// Library/POUs/Read/MC_ReadToolData/Structures/ReadToolDataParCmd
{attribute 'pack_mode' := '1'} 
// ------------------------------------------------------------------------- 
//  SRCI Robot Library                                                
// ------------------------------------------------------------------------- 
//                                                                           
//  Object:      ReadToolDataParCmd                                       
//  Author:      Thorsten Brach                                                
//  Date:        2024-08-09
//
//  Description:                                              
//   
//                                                                           
//  Copyright: 
//    (C) 2024 Thorsten Brach. All rights reserved                                                                                                                                            
//             Licensed under the LGPL-3.0 license.
//                                                                           
//  Disclaimer:                                                                           
//    This project is provided without any guarantee and can be used for   
//    private and commercial purposes. Any use is at the user’s 
//    own risk and responsibility.
//
// -------------------------------------------------------------------------
TYPE ReadToolDataParCmd :
STRUCT
  /// Tool index
  /// • -1: Currently used tool on RC
  /// •  0: Flange -  Not possible to change
  /// • 1 (default)..254: Tool Frame
  ToolNo             : INT;
END_STRUCT
END_TYPE

// Library/POUs/Read/MC_ReadToolData/Structures/ReadToolDataRecvData
{attribute 'pack_mode' := '1'} 
// ------------------------------------------------------------------------- 
//  SRCI Robot Library                                                
// ------------------------------------------------------------------------- 
//                                                                           
//  Object:      ReadToolDataRecvData                                       
//  Author:      Thorsten Brach                                                
//  Date:        2024-08-09
//
//  Description:                                              
//   
//                                                                           
//  Copyright: 
//    (C) 2024 Thorsten Brach. All rights reserved                                                                                                                                            
//             Licensed under the LGPL-3.0 license.
//                                                                           
//  Disclaimer:                                                                           
//    This project is provided without any guarantee and can be used for   
//    private and commercial purposes. Any use is at the user’s 
//    own risk and responsibility.
//
// -------------------------------------------------------------------------
TYPE ReadToolDataRecvData EXTENDS RspHeader :
STRUCT
  /// Reserve
  Reserve       : BYTE;
  /// Tool index
  ToolNoReturn  : USINT;
  /// Tool data (see chapter 5.5.6.3)
  ToolData      : ToolData;
  /// ToDo
  DataChanged   : BOOL;
END_STRUCT
END_TYPE

// Library/POUs/Read/MC_ReadToolData/Structures/ReadToolDataSendData
{attribute 'pack_mode' := '1'}
// ------------------------------------------------------------------------- 
//  SRCI Robot Library                                                
// ------------------------------------------------------------------------- 
//                                                                           
//  Object:      ReadToolDataSendData                                       
//  Author:      Thorsten Brach                                                
//  Date:        2024-08-09
//
//  Description:                                              
//   
//                                                                           
//  Copyright: 
//    (C) 2024 Thorsten Brach. All rights reserved                                                                                                                                            
//             Licensed under the LGPL-3.0 license.
//                                                                           
//  Disclaimer:                                                                           
//    This project is provided without any guarantee and can be used for   
//    private and commercial purposes. Any use is at the user’s 
//    own risk and responsibility.
//
// -------------------------------------------------------------------------
TYPE ReadToolDataSendData EXTENDS CmdHeader: 
STRUCT
  /// Tool index
  /// • -1: Currently used tool on RC
  /// •  0: Flange -  Not possible to change
  /// • 1 (default)..254: Tool Frame
  ToolNo             : INT;
END_STRUCT
END_TYPE

// Library/POUs/SearchHardstop/MC_SearchHardStop/Structures/SearchHardStopOutCmd
{attribute 'pack_mode' := '1'} 
// ------------------------------------------------------------------------- 
//  SRCI Robot Library                                                
// ------------------------------------------------------------------------- 
//                                                                           
//  Object:      SearchHardStopOutCmd                                       
//  Author:      Thorsten Brach                                                
//  Date:        2024-08-01
//
//  Description:                                              
//   
//                                                                           
//  Copyright: 
//    (C) 2024 Thorsten Brach. All rights reserved                                                                                                                                            
//             Licensed under the LGPL-3.0 license.
//                                                                           
//  Disclaimer:                                                                           
//    This project is provided without any guarantee and can be used for   
//    private and commercial purposes. Any use is at the user’s 
//    own risk and responsibility.
//
// -------------------------------------------------------------------------
TYPE SearchHardStopOutCmd :
STRUCT
  /// Distance-to-go of the current job.
  /// • -1: No valid value because move command is not yet active (valid values are pending) or not supported by RC
  /// • >0: Actual distance between current and target position
  /// •  0: Target position reached
  RemainingDistance  : REAL;
  /// Percentage of already traversed distance of current job.
  /// If not supported : • -1
  Progress           : REAL;
  /// The robot arm has detected an obstruction and stopped the movement
  InClamping         : BOOL;  
END_STRUCT
END_TYPE

// Library/POUs/SearchHardstop/MC_SearchHardStop/Structures/SearchHardStopParCmd
{attribute 'pack_mode' := '1'} 
// ------------------------------------------------------------------------- 
//  SRCI Robot Library                                                
// ------------------------------------------------------------------------- 
//                                                                           
//  Object:      SearchHardStopParCmd                                       
//  Author:      Thorsten Brach                                                
//  Date:        2024-08-01
//
//  Description:                                              
//   
//                                                                           
//  Copyright: 
//    (C) 2024 Thorsten Brach. All rights reserved                                                                                                                                            
//             Licensed under the LGPL-3.0 license.
//                                                                           
//  Disclaimer:                                                                           
//    This project is provided without any guarantee and can be used for   
//    private and commercial purposes. Any use is at the user’s 
//    own risk and responsibility.
//
// -------------------------------------------------------------------------
TYPE SearchHardStopParCmd :
STRUCT
  /// Absolute target coordinates in the selected coordinate system (see input parameters ToolNo and FrameNo)
  Position           : RobotCartesianPosition;
  /// Defines the type of collision detection, which parameter should be observed
  DetectionMode      : DetectionMode;
  /// Additional parameter for the detection of an end position. Defines the limits for seven joints, 
  /// where the robot stops when one of the limits is reached. Unit is depending on the "DetectionMode":
  /// • Torque (default) [Nm]  - Only positive values accepted
  /// • Force [N]              - Only positive values accepted
  /// • Electrical current [A] - Only positive values accepted
  /// • Following Error [mm]   - >0: Robot stops when the following error reached positive limit
  ///                          - <0: Robot stops when the following error reaches the negative limit
  DetectionVector    : ARRAY [0..5] OF REAL;
  /// TCP velocity in % of nominal velocity
  /// •  <0%: (default) - Use default velocity
  /// •   0%:           - Use internal minimal velocity
  /// • 100%:           - Use maximal reference velocity
  /// See chapter 5.5.7 Robot dynamics
  VelocityRate       : REAL;
  /// Acceleration for movement in % of nominal acceleration
  /// •  <0%: (default) - Use default acceleration
  /// •   0%:           - Use internal minimal acceleration
  /// • 100%:           - Use maximal reference acceleration
  /// See chapter 5.5.7 Robot dynamics
  AccelerationRate   : REAL;
  /// Deceleration for movement in % of nominal deceleration
  /// •  <0%: (default) - Use default deceleration 
  /// •   0%:           - Use internal minimal deceleration
  /// • 100%:           - Use maximal reference deceleration
  /// See chapter 5.5.7 Robot dynamics
  DecelerationRate   : REAL;
  /// Jerk of the movement in % of nominal jerk
  /// •  <0%: (default) - Use default jerk
  /// •   0%:           - Use internal minimal jerk
  /// • 100%:           - Use maximal reference jerk
  /// See chapter 5.5.7 Robot dynamics
  JerkRate           : REAL;
  /// Index of tool
  /// •      0: Flange (default)
  /// • 1..254: Tool frames
  ToolNo             : USINT;
  /// Index of frame
  /// •      0: WCS (default)
  /// • 1..254: User frames
  FrameNo            : USINT;
  /// Parameter to describe how the orientation axes (RX, RY, RZ) will be interpolated during the movement
  OriMode            : OriMode;
  /// Defines the usage of the config byte inside the position according to Table 6-238
  ConfigMode         : ArmConfigParameter;
  /// Defines the usage of the TurnNumber byte inside the position.
  TurnMode           : TurnMode;
  /// Set TRUE to allow manipulation of this move command through superimposing functions.
  /// For more information see chapter 5.5.9.5
  Manipulation       : BOOL;
END_STRUCT
END_TYPE

// Library/POUs/SearchHardstop/MC_SearchHardStop/Structures/SearchHardStopRecvData
{attribute 'pack_mode' := '1'} 
// ------------------------------------------------------------------------- 
//  SRCI Robot Library                                                
// ------------------------------------------------------------------------- 
//                                                                           
//  Object:      SearchHardStopRecvData                                       
//  Author:      Thorsten Brach                                                
//  Date:        2024-08-01
//
//  Description:                                              
//   
//                                                                           
//  Copyright: 
//    (C) 2024 Thorsten Brach. All rights reserved                                                                                                                                            
//             Licensed under the LGPL-3.0 license.
//                                                                           
//  Disclaimer:                                                                           
//    This project is provided without any guarantee and can be used for   
//    private and commercial purposes. Any use is at the user’s 
//    own risk and responsibility.
//
// -------------------------------------------------------------------------
TYPE SearchHardStopRecvData EXTENDS RspHeader :
STRUCT
  /// Percentage of already traversed distance of current job.
  /// If not supported : • -1
  Progress           : UINT;
  /// Distance-to-go of the current job.
  /// • -1: No valid value because move command is not yet active (valid values are pending) or not supported by RC
  /// • >0: Actual distance between current and target position
  /// •  0: Target position reached
  RemainingDistance  : REAL;
  /// The robot arm has detected an obstruction and stopped the movement
  InClamping         : BOOL;  
END_STRUCT
END_TYPE

// Library/POUs/SearchHardstop/MC_SearchHardStop/Structures/SearchHardStopSendData
{attribute 'pack_mode' := '1'}
// ------------------------------------------------------------------------- 
//  SRCI Robot Library                                                
// ------------------------------------------------------------------------- 
//                                                                           
//  Object:      SearchHardStopSendData                                       
//  Author:      Thorsten Brach                                                
//  Date:        2024-08-01
//
//  Description:                                              
//   
//                                                                           
//  Copyright: 
//    (C) 2024 Thorsten Brach. All rights reserved                                                                                                                                            
//             Licensed under the LGPL-3.0 license.
//                                                                           
//  Disclaimer:                                                                           
//    This project is provided without any guarantee and can be used for   
//    private and commercial purposes. Any use is at the user’s 
//    own risk and responsibility.
//
// -------------------------------------------------------------------------
TYPE SearchHardStopSendData EXTENDS CmdHeader: 
STRUCT
  /// TCP velocity in % of nominal velocity
  /// •  <0%: (default) - Use default velocity
  /// •   0%:           - Use internal minimal velocity
  /// • 100%:           - Use maximal reference velocity
  /// See chapter 5.5.7 Robot dynamics
  VelocityRate       : UINT;
  /// Acceleration for movement in % of nominal acceleration
  /// •  <0%: (default) - Use default acceleration
  /// •   0%:           - Use internal minimal acceleration
  /// • 100%:           - Use maximal reference acceleration
  /// See chapter 5.5.7 Robot dynamics
  AccelerationRate   : UINT;
  /// Deceleration for movement in % of nominal deceleration
  /// •  <0%: (default) - Use default deceleration 
  /// •   0%:           - Use internal minimal deceleration
  /// • 100%:           - Use maximal reference deceleration
  /// See chapter 5.5.7 Robot dynamics
  DecelerationRate   : UINT;
  /// Jerk of the movement in % of nominal jerk
  /// •  <0%: (default) - Use default jerk
  /// •   0%:           - Use internal minimal jerk
  /// • 100%:           - Use maximal reference jerk
  /// See chapter 5.5.7 Robot dynamics
  JerkRate           : UINT;
  /// Index of tool
  /// •      0: Flange (default)
  /// • 1..254: Tool frames
  ToolNo             : USINT;
  /// Index of frame
  /// •      0: WCS (default)
  /// • 1..254: User frames
  FrameNo            : USINT;
  /// Absolute target coordinates in the selected coordinate system (see input parameters ToolNo and FrameNo)
  Position           : RobotCartesianPosition;
  /// Parameter to describe how the orientation axes (RX, RY, RZ) will be interpolated during the movement
  OriMode            : USINT;
  /// Defines the type of collision detection, which parameter should be observed
  DetectionMode      : USINT;
  /// Set TRUE to allow manipulation of this move command through superimposing functions.
  /// For more information see chapter 5.5.9.5
  Manipulation       : BOOL;
  /// Reserve
  Reserve            : BYTE;
  /// Additional parameter for the detection of an end position. Defines the limits for seven joints, 
  /// where the robot stops when one of the limits is reached. Unit is depending on the "DetectionMode":
  /// • Torque (default) [Nm]  - Only positive values accepted
  /// • Force [N]              - Only positive values accepted
  /// • Electrical current [A] - Only positive values accepted
  /// • Following Error [mm]   - >0: Robot stops when the following error reached positive limit
  ///                          - <0: Robot stops when the following error reaches the negative limit
  DetectionVector    : ARRAY [0..5] OF REAL;
  /// Defines the usage of the config byte inside the position according to Table 6-238
  ConfigMode         : ARRAY [0..1] OF BYTE;
  /// Defines the usage of the TurnNumber byte inside the position.
  TurnMode           : USINT;
END_STRUCT
END_TYPE

// Library/POUs/SearchHardstop/MC_SearchHardStopJ/Structures/SearchHardStopJOutCmd
{attribute 'pack_mode' := '1'} 
// ------------------------------------------------------------------------- 
//  SRCI Robot Library                                                
// ------------------------------------------------------------------------- 
//                                                                           
//  Object:      SearchHardStopOutCmd                                       
//  Author:      Thorsten Brach                                                
//  Date:        2024-08-01
//
//  Description:                                              
//   
//                                                                           
//  Copyright: 
//    (C) 2024 Thorsten Brach. All rights reserved                                                                                                                                            
//             Licensed under the LGPL-3.0 license.
//                                                                           
//  Disclaimer:                                                                           
//    This project is provided without any guarantee and can be used for   
//    private and commercial purposes. Any use is at the user’s 
//    own risk and responsibility.
//
// -------------------------------------------------------------------------
TYPE SearchHardStopJOutCmd :
STRUCT
  /// Distance-to-go of the current job.
  /// • -1: No valid value because move command is not yet active (valid values are pending) or not supported by RC
  /// • >0: Actual distance between current and target position
  /// •  0: Target position reached
  RemainingDistance  : REAL;
  /// Percentage of already traversed distance of current job.
  /// If not supported : • -1
  Progress           : REAL;
  /// The robot arm has detected an obstruction and stopped the movement
  InClamping         : BOOL;  
END_STRUCT
END_TYPE

// Library/POUs/SearchHardstop/MC_SearchHardStopJ/Structures/SearchHardStopJParCmd
{attribute 'pack_mode' := '1'} 
// ------------------------------------------------------------------------- 
//  SRCI Robot Library                                                
// ------------------------------------------------------------------------- 
//                                                                           
//  Object:      SearchHardStopParCmd                                       
//  Author:      Thorsten Brach                                                
//  Date:        2024-08-01
//
//  Description:                                              
//   
//                                                                           
//  Copyright: 
//    (C) 2024 Thorsten Brach. All rights reserved                                                                                                                                            
//             Licensed under the LGPL-3.0 license.
//                                                                           
//  Disclaimer:                                                                           
//    This project is provided without any guarantee and can be used for   
//    private and commercial purposes. Any use is at the user’s 
//    own risk and responsibility.
//
// -------------------------------------------------------------------------
TYPE SearchHardStopJParCmd :
STRUCT
  /// Absolute end position of the robot in Joint position.
  JointPosition      : RobotJointPosition;
  /// Defines the type of collision detection, which parameter should be observed
  DetectionMode      : DetectionMode;
  /// Additional parameter for the detection of an end position. Defines the limits for seven joints, 
  /// where the robot stops when one of the limits is reached. Unit is depending on the "DetectionMode":
  /// • Torque (default) [Nm]  - Only positive values accepted
  /// • Force [N]              - Only positive values accepted
  /// • Electrical current [A] - Only positive values accepted
  /// • Following Error [mm]   - >0: Robot stops when the following error reached positive limit
  ///                          - <0: Robot stops when the following error reaches the negative limit
  DetectionVector    : ARRAY [0..5] OF REAL;
  /// TCP velocity in % of nominal velocity
  /// •  <0%: (default) - Use default velocity
  /// •   0%:           - Use internal minimal velocity
  /// • 100%:           - Use maximal reference velocity
  /// See chapter 5.5.7 Robot dynamics
  VelocityRate       : REAL;
  /// Acceleration for movement in % of nominal acceleration
  /// •  <0%: (default) - Use default acceleration
  /// •   0%:           - Use internal minimal acceleration
  /// • 100%:           - Use maximal reference acceleration
  /// See chapter 5.5.7 Robot dynamics
  AccelerationRate   : REAL;
  /// Deceleration for movement in % of nominal deceleration
  /// •  <0%: (default) - Use default deceleration 
  /// •   0%:           - Use internal minimal deceleration
  /// • 100%:           - Use maximal reference deceleration
  /// See chapter 5.5.7 Robot dynamics
  DecelerationRate   : REAL;
  /// Jerk of the movement in % of nominal jerk
  /// •  <0%: (default) - Use default jerk
  /// •   0%:           - Use internal minimal jerk
  /// • 100%:           - Use maximal reference jerk
  /// See chapter 5.5.7 Robot dynamics
  JerkRate           : REAL;
  /// Index of tool
  /// •      0: Flange (default)
  /// • 1..254: Tool frames
  ToolNo             : USINT;
  /// Set TRUE to allow manipulation of this move command through superimposing functions.
  /// For more information see chapter 5.5.9.5
  Manipulation       : BOOL;
END_STRUCT
END_TYPE

// Library/POUs/SearchHardstop/MC_SearchHardStopJ/Structures/SearchHardStopJRecvData
{attribute 'pack_mode' := '1'} 
// ------------------------------------------------------------------------- 
//  SRCI Robot Library                                                
// ------------------------------------------------------------------------- 
//                                                                           
//  Object:      SearchHardStopRecvData                                       
//  Author:      Thorsten Brach                                                
//  Date:        2024-08-01
//
//  Description:                                              
//   
//                                                                           
//  Copyright: 
//    (C) 2024 Thorsten Brach. All rights reserved                                                                                                                                            
//             Licensed under the LGPL-3.0 license.
//                                                                           
//  Disclaimer:                                                                           
//    This project is provided without any guarantee and can be used for   
//    private and commercial purposes. Any use is at the user’s 
//    own risk and responsibility.
//
// -------------------------------------------------------------------------
TYPE SearchHardStopJRecvData EXTENDS RspHeader :
STRUCT
  /// Percentage of already traversed distance of current job.
  /// If not supported : • -1
  Progress           : UINT;
  /// Distance-to-go of the current job.
  /// • -1: No valid value because move command is not yet active (valid values are pending) or not supported by RC
  /// • >0: Actual distance between current and target position
  /// •  0: Target position reached
  RemainingDistance  : REAL;
  /// The robot arm has detected an obstruction and stopped the movement
  InClamping         : BOOL;  
END_STRUCT
END_TYPE

// Library/POUs/SearchHardstop/MC_SearchHardStopJ/Structures/SearchHardStopJSendData
{attribute 'pack_mode' := '1'}
// ------------------------------------------------------------------------- 
//  SRCI Robot Library                                                
// ------------------------------------------------------------------------- 
//                                                                           
//  Object:      SearchHardStopSendData                                       
//  Author:      Thorsten Brach                                                
//  Date:        2024-08-01
//
//  Description:                                              
//   
//                                                                           
//  Copyright: 
//    (C) 2024 Thorsten Brach. All rights reserved                                                                                                                                            
//             Licensed under the LGPL-3.0 license.
//                                                                           
//  Disclaimer:                                                                           
//    This project is provided without any guarantee and can be used for   
//    private and commercial purposes. Any use is at the user’s 
//    own risk and responsibility.
//
// -------------------------------------------------------------------------
TYPE SearchHardStopJSendData EXTENDS CmdHeader: 
STRUCT
  /// TCP velocity in % of nominal velocity
  /// •  <0%: (default) - Use default velocity
  /// •   0%:           - Use internal minimal velocity
  /// • 100%:           - Use maximal reference velocity
  /// See chapter 5.5.7 Robot dynamics
  VelocityRate       : UINT;
  /// Acceleration for movement in % of nominal acceleration
  /// •  <0%: (default) - Use default acceleration
  /// •   0%:           - Use internal minimal acceleration
  /// • 100%:           - Use maximal reference acceleration
  /// See chapter 5.5.7 Robot dynamics
  AccelerationRate   : UINT;
  /// Deceleration for movement in % of nominal deceleration
  /// •  <0%: (default) - Use default deceleration 
  /// •   0%:           - Use internal minimal deceleration
  /// • 100%:           - Use maximal reference deceleration
  /// See chapter 5.5.7 Robot dynamics
  DecelerationRate   : UINT;
  /// Jerk of the movement in % of nominal jerk
  /// •  <0%: (default) - Use default jerk
  /// •   0%:           - Use internal minimal jerk
  /// • 100%:           - Use maximal reference jerk
  /// See chapter 5.5.7 Robot dynamics
  JerkRate           : UINT;
  /// Absolute end position of the robot in Joint position.
  JointPosition      : RobotJointPosition;
  /// Parameter to describe how the orientation axes (RX, RY, RZ) will be interpolated during the movement
  OriMode            : USINT;
  /// Defines the type of collision detection, which parameter should be observed
  DetectionMode      : USINT;
  /// Set TRUE to allow manipulation of this move command through superimposing functions.
  /// For more information see chapter 5.5.9.5
  Manipulation       : BOOL;
  /// Reserve
  Reserve            : BYTE;
  /// Additional parameter for the detection of an end position. Defines the limits for seven joints, 
  /// where the robot stops when one of the limits is reached. Unit is depending on the "DetectionMode":
  /// • Torque (default) [Nm]  - Only positive values accepted
  /// • Force [N]              - Only positive values accepted
  /// • Electrical current [A] - Only positive values accepted
  /// • Following Error [mm]   - >0: Robot stops when the following error reached positive limit
  ///                          - <0: Robot stops when the following error reaches the negative limit
  DetectionVector    : ARRAY [0..5] OF REAL;
END_STRUCT
END_TYPE

// Library/POUs/Spline/MC_CreateSpline/Structures/CreateSplineOutCmd
{attribute 'pack_mode' := '1'} 
// ------------------------------------------------------------------------- 
//  SRCI Robot Library                                                
// ------------------------------------------------------------------------- 
//                                                                           
//  Object:      CreateSplineOutCmd                                       
//  Author:      Thorsten Brach                                                
//  Date:        2024-08-01
//
//  Description:                                              
//   
//                                                                           
//  Copyright: 
//    (C) 2024 Thorsten Brach. All rights reserved                                                                                                                                            
//             Licensed under the LGPL-3.0 license.
//                                                                           
//  Disclaimer:                                                                           
//    This project is provided without any guarantee and can be used for   
//    private and commercial purposes. Any use is at the user’s 
//    own risk and responsibility.
//
// -------------------------------------------------------------------------
TYPE CreateSplineOutCmd :
STRUCT
END_STRUCT
END_TYPE

// Library/POUs/Spline/MC_CreateSpline/Structures/CreateSplineParCmd
{attribute 'pack_mode' := '1'} 
// ------------------------------------------------------------------------- 
//  SRCI Robot Library                                                
// ------------------------------------------------------------------------- 
//                                                                           
//  Object:      CreateSplineParCmd                                       
//  Author:      Thorsten Brach                                                
//  Date:        2024-08-01
//
//  Description:                                              
//   
//                                                                           
//  Copyright: 
//    (C) 2024 Thorsten Brach. All rights reserved                                                                                                                                            
//             Licensed under the LGPL-3.0 license.
//                                                                           
//  Disclaimer:                                                                           
//    This project is provided without any guarantee and can be used for   
//    private and commercial purposes. Any use is at the user’s 
//    own risk and responsibility.
//
// -------------------------------------------------------------------------
TYPE CreateSplineParCmd :
STRUCT
  /// Define the method to calculate the path trajectory for the spline movement
  Mode            : SplineMode;
  /// Index of the spline trajectory to be created
  SplineID        : SINT;
  /// Contains all data relevant to the spline trajectory
  /// • Cartesian position
  /// • Coordinate systems
  /// • Dynamic parameters
  /// For more information refer to chapter 5.5.13.3
  SplineData      : ARRAY[1..RobotLibraryParameter.SPLINE_DATA_MAX] OF SplineData;
END_STRUCT
END_TYPE

// Library/POUs/Spline/MC_CreateSpline/Structures/CreateSplineRecvData
{attribute 'pack_mode' := '1'} 
// ------------------------------------------------------------------------- 
//  SRCI Robot Library                                                
// ------------------------------------------------------------------------- 
//                                                                           
//  Object:      CreateSplineRecvData                                       
//  Author:      Thorsten Brach                                                
//  Date:        2024-08-01
//
//  Description:                                              
//   
//                                                                           
//  Copyright: 
//    (C) 2024 Thorsten Brach. All rights reserved                                                                                                                                            
//             Licensed under the LGPL-3.0 license.
//                                                                           
//  Disclaimer:                                                                           
//    This project is provided without any guarantee and can be used for   
//    private and commercial purposes. Any use is at the user’s 
//    own risk and responsibility.
//
// -------------------------------------------------------------------------
TYPE CreateSplineRecvData EXTENDS RspHeader :
STRUCT
END_STRUCT
END_TYPE

// Library/POUs/Spline/MC_CreateSpline/Structures/CreateSplineSendData
{attribute 'pack_mode' := '1'}
// ------------------------------------------------------------------------- 
//  SRCI Robot Library                                                
// ------------------------------------------------------------------------- 
//                                                                           
//  Object:      CreateSplineSendData                                       
//  Author:      Thorsten Brach                                                
//  Date:        2024-08-01
//
//  Description:                                              
//   
//                                                                           
//  Copyright: 
//    (C) 2024 Thorsten Brach. All rights reserved                                                                                                                                            
//             Licensed under the LGPL-3.0 license.
//                                                                           
//  Disclaimer:                                                                           
//    This project is provided without any guarantee and can be used for   
//    private and commercial purposes. Any use is at the user’s 
//    own risk and responsibility.
//
// -------------------------------------------------------------------------
TYPE CreateSplineSendData EXTENDS CmdHeader: 
STRUCT
  /// Define the method to calculate the path trajectory for the spline movement
  Mode            : UINT;
  /// Index of the spline trajectory to be created
  SplineID        : SINT;
  /// Contains all data relevant to the spline trajectory
  /// • Cartesian position
  /// • Coordinate systems
  /// • Dynamic parameters
  /// For more information refer to chapter 5.5.13.3
  SplineData      : ARRAY[1..RobotLibraryParameter.SPLINE_DATA_MAX] OF SplineDataSend;
END_STRUCT
END_TYPE

// Library/POUs/Spline/MC_DeleteSpline/Structures/DeleteSplineOutCmd
{attribute 'pack_mode' := '1'} 
// ------------------------------------------------------------------------- 
//  SRCI Robot Library                                                
// ------------------------------------------------------------------------- 
//                                                                           
//  Object:      DeleteSplineOutCmd                                       
//  Author:      Thorsten Brach                                                
//  Date:        2024-08-01
//
//  Description:                                              
//   
//                                                                           
//  Copyright: 
//    (C) 2024 Thorsten Brach. All rights reserved                                                                                                                                            
//             Licensed under the LGPL-3.0 license.
//                                                                           
//  Disclaimer:                                                                           
//    This project is provided without any guarantee and can be used for   
//    private and commercial purposes. Any use is at the user’s 
//    own risk and responsibility.
//
// -------------------------------------------------------------------------
TYPE DeleteSplineOutCmd :
STRUCT
END_STRUCT
END_TYPE

// Library/POUs/Spline/MC_DeleteSpline/Structures/DeleteSplineParCmd
{attribute 'pack_mode' := '1'} 
// ------------------------------------------------------------------------- 
//  SRCI Robot Library                                                
// ------------------------------------------------------------------------- 
//                                                                           
//  Object:      DeleteSplineParCmd                                       
//  Author:      Thorsten Brach                                                
//  Date:        2024-08-01
//
//  Description:                                              
//   
//                                                                           
//  Copyright: 
//    (C) 2024 Thorsten Brach. All rights reserved                                                                                                                                            
//             Licensed under the LGPL-3.0 license.
//                                                                           
//  Disclaimer:                                                                           
//    This project is provided without any guarantee and can be used for   
//    private and commercial purposes. Any use is at the user’s 
//    own risk and responsibility.
//
// -------------------------------------------------------------------------
TYPE DeleteSplineParCmd :
STRUCT
  /// Index of the spline trajectory to be deleted
  SplineID        : SINT;
END_STRUCT
END_TYPE

// Library/POUs/Spline/MC_DeleteSpline/Structures/DeleteSplineRecvData
{attribute 'pack_mode' := '1'} 
// ------------------------------------------------------------------------- 
//  SRCI Robot Library                                                
// ------------------------------------------------------------------------- 
//                                                                           
//  Object:      DeleteSplineRecvData                                       
//  Author:      Thorsten Brach                                                
//  Date:        2024-08-01
//
//  Description:                                              
//   
//                                                                           
//  Copyright: 
//    (C) 2024 Thorsten Brach. All rights reserved                                                                                                                                            
//             Licensed under the LGPL-3.0 license.
//                                                                           
//  Disclaimer:                                                                           
//    This project is provided without any guarantee and can be used for   
//    private and commercial purposes. Any use is at the user’s 
//    own risk and responsibility.
//
// -------------------------------------------------------------------------
TYPE DeleteSplineRecvData EXTENDS RspHeader :
STRUCT
END_STRUCT
END_TYPE

// Library/POUs/Spline/MC_DeleteSpline/Structures/DeleteSplineSendData
{attribute 'pack_mode' := '1'}
// ------------------------------------------------------------------------- 
//  SRCI Robot Library                                                
// ------------------------------------------------------------------------- 
//                                                                           
//  Object:      DeleteSplineSendData                                       
//  Author:      Thorsten Brach                                                
//  Date:        2024-08-01
//
//  Description:                                              
//   
//                                                                           
//  Copyright: 
//    (C) 2024 Thorsten Brach. All rights reserved                                                                                                                                            
//             Licensed under the LGPL-3.0 license.
//                                                                           
//  Disclaimer:                                                                           
//    This project is provided without any guarantee and can be used for   
//    private and commercial purposes. Any use is at the user’s 
//    own risk and responsibility.
//
// -------------------------------------------------------------------------
TYPE DeleteSplineSendData EXTENDS CmdHeader: 
STRUCT
  /// Index of the spline trajectory to be deleted
  SplineID        : SINT;
END_STRUCT
END_TYPE

// Library/POUs/Spline/MC_DynamicSpline/Structures/DynamicSplineOutCmd
{attribute 'pack_mode' := '1'} 
// ------------------------------------------------------------------------- 
//  SRCI Robot Library                                                
// ------------------------------------------------------------------------- 
//                                                                           
//  Object:      DynamicSplineOutCmd                                       
//  Author:      Thorsten Brach                                                
//  Date:        2024-08-01
//
//  Description:                                              
//   
//                                                                           
//  Copyright: 
//    (C) 2024 Thorsten Brach. All rights reserved                                                                                                                                            
//             Licensed under the LGPL-3.0 license.
//                                                                           
//  Disclaimer:                                                                           
//    This project is provided without any guarantee and can be used for   
//    private and commercial purposes. Any use is at the user’s 
//    own risk and responsibility.
//
// -------------------------------------------------------------------------
TYPE DynamicSplineOutCmd :
STRUCT
  /// Distance-to-go of the current job.
  /// • -1: No valid value because move command is not yet active (valid values are pending) or not supported by RC
  /// • >0: Actual distance between current and target position
  /// •  0: Target position reached 
  RemainingDistance  : REAL;
  /// Percentage of already traversed distance of actual segment of spline trajectory.
  /// If not supported: -1
  SegmentProgress    : REAL;
  /// Number of buffered, consecutive segments of spline trajectory. 
  Buffered           : INT;
  /// Number of calculated, consecutive segments of spline trajectory. Already calculated segments can no longer be modified.
  Calculated         : INT;
  /// Index of the currently active segment of spline data set.
  ActiveIndex        : SINT;  
  /// Spline movement has been finished successfully. New SplineData will start a new spline movement.
  TrajectoryCompleted: BOOL;  
END_STRUCT
END_TYPE

// Library/POUs/Spline/MC_DynamicSpline/Structures/DynamicSplineParCmd
{attribute 'pack_mode' := '1'} 
// ------------------------------------------------------------------------- 
//  SRCI Robot Library                                                
// ------------------------------------------------------------------------- 
//                                                                           
//  Object:      DynamicSplineParCmd                                       
//  Author:      Thorsten Brach                                                
//  Date:        2024-08-01
//
//  Description:                                              
//   
//                                                                           
//  Copyright: 
//    (C) 2024 Thorsten Brach. All rights reserved                                                                                                                                            
//             Licensed under the LGPL-3.0 license.
//                                                                           
//  Disclaimer:                                                                           
//    This project is provided without any guarantee and can be used for   
//    private and commercial purposes. Any use is at the user’s 
//    own risk and responsibility.
//
// -------------------------------------------------------------------------
TYPE DynamicSplineParCmd :
STRUCT
  /// Define the method to calculate the path trajectory for the spline movement
  Mode               : SplineMode;
  /// Parameter which determines the transition behavior at the end of the movement to be sent to the next command. 
  /// The user can choose a transition type between exact stop and different blend possibilities.
  BlendingMode       : BlendingMode;
  /// Additional parameter for the blending mode, to define i.e. velocity limit (%) or blending radius
  /// • [0]: default 10
  /// • [1]: default 0
  BlendingParameter  : ARRAY [0..1] OF REAL;
  /// Parameter is used if it is greater than 0 (default):
  /// • Velocity input is ignored
  /// • Parameter defines the time for the movement to reach the target position 
  /// Error is sent by the RC, if the time cannot be kept.
  MoveTime           : TIME;
  /// Contains all data relevant to the spline trajectory
  /// • Cartesian position
  /// • Coordinate systems
  /// • Dynamic parameters
  /// For more information refer to chapter 5.5.13.3
  SplineData         : ARRAY[1..RobotLibraryParameter.SPLINE_DATA_MAX] OF SplineData;
  /// Starts calculation and spline motion when equal or greater to number of buffered spline positions
  StartPosition      : INT; 
END_STRUCT
END_TYPE

// Library/POUs/Spline/MC_DynamicSpline/Structures/DynamicSplineRecvData
{attribute 'pack_mode' := '1'} 
// ------------------------------------------------------------------------- 
//  SRCI Robot Library                                                
// ------------------------------------------------------------------------- 
//                                                                           
//  Object:      DynamicSplineRecvData                                       
//  Author:      Thorsten Brach                                                
//  Date:        2024-08-01
//
//  Description:                                              
//   
//                                                                           
//  Copyright: 
//    (C) 2024 Thorsten Brach. All rights reserved                                                                                                                                            
//             Licensed under the LGPL-3.0 license.
//                                                                           
//  Disclaimer:                                                                           
//    This project is provided without any guarantee and can be used for   
//    private and commercial purposes. Any use is at the user’s 
//    own risk and responsibility.
//
// -------------------------------------------------------------------------
TYPE DynamicSplineRecvData EXTENDS RspHeader :
STRUCT
  /// Distance-to-go of the current job.
  /// • -1: No valid value because move command is not yet active (valid values are pending) or not supported by RC
  /// • >0: Actual distance between current and target position
  /// •  0: Target position reached 
  RemainingDistance  : REAL;
  /// Percentage of already traversed distance of actual segment of spline trajectory.
  /// If not supported: -1
  SegmentProgress    : REAL;
  /// Number of buffered, consecutive segments of spline trajectory. 
  Buffered           : INT;
  /// Number of calculated, consecutive segments of spline trajectory. Already calculated segments can no longer be modified.
  Calculated         : INT;
  /// Index of the currently active segment of spline data set.
  ActiveIndex        : SINT;  
  /// Spline movement has been finished successfully. New SplineData will start a new spline movement.
  TrajectoryCompleted: BOOL;  
END_STRUCT
END_TYPE

// Library/POUs/Spline/MC_DynamicSpline/Structures/DynamicSplineSendData
{attribute 'pack_mode' := '1'}
// ------------------------------------------------------------------------- 
//  SRCI Robot Library                                                
// ------------------------------------------------------------------------- 
//                                                                           
//  Object:      DynamicSplineSendData                                       
//  Author:      Thorsten Brach                                                
//  Date:        2024-08-01
//
//  Description:                                              
//   
//                                                                           
//  Copyright: 
//    (C) 2024 Thorsten Brach. All rights reserved                                                                                                                                            
//             Licensed under the LGPL-3.0 license.
//                                                                           
//  Disclaimer:                                                                           
//    This project is provided without any guarantee and can be used for   
//    private and commercial purposes. Any use is at the user’s 
//    own risk and responsibility.
//
// -------------------------------------------------------------------------
TYPE DynamicSplineSendData EXTENDS CmdHeader: 
STRUCT
  /// Define the method to calculate the path trajectory for the spline movement
  Mode               : UINT;
  /// Parameter which determines the transition behavior at the end of the movement to be sent to the next command. 
  /// The user can choose a transition type between exact stop and different blend possibilities.
  BlendingMode       : USINT;
  /// Additional parameter for the blending mode, to define i.e. velocity limit (%) or blending radius
  /// • [0]: default 10
  /// • [1]: default 0
  BlendingParameter  : ARRAY [0..1] OF REAL;
  /// Parameter is used if it is greater than 0 (default):
  /// • Velocity input is ignored
  /// • Parameter defines the time for the movement to reach the target position 
  /// Error is sent by the RC, if the time cannot be kept.
  MoveTime           : UINT;
  /// Starts calculation and spline motion when equal or greater to number of buffered spline positions
  StartPosition      : INT; 
  /// Contains all data relevant to the spline trajectory
  /// • Cartesian position
  /// • Coordinate systems
  /// • Dynamic parameters
  /// For more information refer to chapter 5.5.13.3
  SplineData         : ARRAY[1..RobotLibraryParameter.SPLINE_DATA_MAX] OF SplineDataSend;
END_STRUCT
END_TYPE

// Library/POUs/Spline/MC_MoveSpline/Structures/MoveSplineOutCmd
{attribute 'pack_mode' := '1'} 
// ------------------------------------------------------------------------- 
//  SRCI Robot Library                                                
// ------------------------------------------------------------------------- 
//                                                                           
//  Object:      MoveSplineOutCmd                                       
//  Author:      Thorsten Brach                                                
//  Date:        2024-08-01
//
//  Description:                                              
//   
//                                                                           
//  Copyright: 
//    (C) 2024 Thorsten Brach. All rights reserved                                                                                                                                            
//             Licensed under the LGPL-3.0 license.
//                                                                           
//  Disclaimer:                                                                           
//    This project is provided without any guarantee and can be used for   
//    private and commercial purposes. Any use is at the user’s 
//    own risk and responsibility.
//
// -------------------------------------------------------------------------
TYPE MoveSplineOutCmd :
STRUCT
  /// Index of the currently active segment of spline data set.
  ActualIndex        : SINT;
  /// Percentage of already traversed distance of current job.
  /// If not supported : • -1
  Progress           : REAL;  
  /// Distance-to-go of the current job.
  /// • -1: No valid value because move command is not yet active (valid values are pending) or not supported by RC
  /// • >0: Actual distance between current and target position
  /// •  0: Target position reached
  RemainingDistance  : REAL;  
END_STRUCT
END_TYPE

// Library/POUs/Spline/MC_MoveSpline/Structures/MoveSplineParCmd
{attribute 'pack_mode' := '1'} 
// ------------------------------------------------------------------------- 
//  SRCI Robot Library                                                
// ------------------------------------------------------------------------- 
//                                                                           
//  Object:      MoveSplineParCmd                                       
//  Author:      Thorsten Brach                                                
//  Date:        2024-08-01
//
//  Description:                                              
//   
//                                                                           
//  Copyright: 
//    (C) 2024 Thorsten Brach. All rights reserved                                                                                                                                            
//             Licensed under the LGPL-3.0 license.
//                                                                           
//  Disclaimer:                                                                           
//    This project is provided without any guarantee and can be used for   
//    private and commercial purposes. Any use is at the user’s 
//    own risk and responsibility.
//
// -------------------------------------------------------------------------
TYPE MoveSplineParCmd :
STRUCT
  /// Index of the spline data set, on which the spline trajectory is based
  SplineID           : SINT;
  /// Parameter which determines the transition behavior at the end of the movement to be sent to the next command. 
  /// The user can choose a transition type between exact stop and different blend possibilities.
  BlendingMode       : BlendingMode;
  /// Additional parameter for the blending mode, to define i.e. velocity limit (%) or blending radius
  /// • [0]: default 10
  /// • [1]: default 0
  BlendingParameter  : ARRAY [0..1] OF REAL;
  /// Parameter is used if it is greater than 0 (default):
  /// • Velocity input is ignored
  /// • Parameter defines the time for the movement to reach the target position 
  /// Error is sent by the RC, if the time cannot be kept.
  MoveTime           : TIME;
END_STRUCT
END_TYPE

// Library/POUs/Spline/MC_MoveSpline/Structures/MoveSplineRecvData
{attribute 'pack_mode' := '1'} 
// ------------------------------------------------------------------------- 
//  SRCI Robot Library                                                
// ------------------------------------------------------------------------- 
//                                                                           
//  Object:      MoveSplineRecvData                                       
//  Author:      Thorsten Brach                                                
//  Date:        2024-08-01
//
//  Description:                                              
//   
//                                                                           
//  Copyright: 
//    (C) 2024 Thorsten Brach. All rights reserved                                                                                                                                            
//             Licensed under the LGPL-3.0 license.
//                                                                           
//  Disclaimer:                                                                           
//    This project is provided without any guarantee and can be used for   
//    private and commercial purposes. Any use is at the user’s 
//    own risk and responsibility.
//
// -------------------------------------------------------------------------
TYPE MoveSplineRecvData EXTENDS RspHeader :
STRUCT
  /// Percentage of already traversed distance of current job.
  /// If not supported : • -1
  Progress          : UINT;
  /// Distance-to-go of the current job.
  /// • -1: No valid value because move command is not yet active (valid values are pending) or not supported by RC
  /// • >0: Actual distance between current and target position
  /// •  0: Target position reached
  RemainingDistance  : REAL;
END_STRUCT
END_TYPE

// Library/POUs/Spline/MC_MoveSpline/Structures/MoveSplineSendData
{attribute 'pack_mode' := '1'}
// ------------------------------------------------------------------------- 
//  SRCI Robot Library                                                
// ------------------------------------------------------------------------- 
//                                                                           
//  Object:      MoveSplineSendData                                       
//  Author:      Thorsten Brach                                                
//  Date:        2024-08-01
//
//  Description:                                              
//   
//                                                                           
//  Copyright: 
//    (C) 2024 Thorsten Brach. All rights reserved                                                                                                                                            
//             Licensed under the LGPL-3.0 license.
//                                                                           
//  Disclaimer:                                                                           
//    This project is provided without any guarantee and can be used for   
//    private and commercial purposes. Any use is at the user’s 
//    own risk and responsibility.
//
// -------------------------------------------------------------------------
TYPE MoveSplineSendData EXTENDS CmdHeader: 
STRUCT
  /// Index of the spline data set, on which the spline trajectory is based
  SplineID           : SINT;
  /// Parameter which determines the transition behavior at the end of the movement to be sent to the next command. 
  /// The user can choose a transition type between exact stop and different blend possibilities.
  BlendingMode       : USINT;
  /// Additional parameter for the blending mode, to define i.e. velocity limit (%) or blending radius
  /// • [0]: default 10
  /// • [1]: default 0
  BlendingParameter  : ARRAY [0..1] OF REAL;
  /// Parameter is used if it is greater than 0 (default):
  /// • Velocity input is ignored
  /// • Parameter defines the time for the movement to reach the target position 
  /// Error is sent by the RC, if the time cannot be kept.
  MoveTime           : UINT;
END_STRUCT
END_TYPE

// Library/POUs/SuperImposing/MC_MoveSuperImposed/Structures/MoveSuperImposedOutCmd
{attribute 'pack_mode' := '1'} 
// ------------------------------------------------------------------------- 
//  SRCI Robot Library                                                
// ------------------------------------------------------------------------- 
//                                                                           
//  Object:      MoveSuperImposedOutCmd                                       
//  Author:      Thorsten Brach                                                
//  Date:        2024-08-01
//
//  Description:                                              
//   
//                                                                           
//  Copyright: 
//    (C) 2024 Thorsten Brach. All rights reserved                                                                                                                                            
//             Licensed under the LGPL-3.0 license.
//                                                                           
//  Disclaimer:                                                                           
//    This project is provided without any guarantee and can be used for   
//    private and commercial purposes. Any use is at the user’s 
//    own risk and responsibility.
//
// -------------------------------------------------------------------------
TYPE MoveSuperImposedOutCmd :
STRUCT
  /// Distance-to-go of the current job.
  /// • -1: No valid value because move command is not yet active (valid values are pending) or not supported by RC
  /// • >0: Actual distance between current and target position
  /// •  0: Target position reached
  RemainingDistance  : REAL;  
  /// Percentage of already traversed distance of current job.
  /// If not supported : • -1
  Progress           : REAL;  
  /// Unique system-generated ID of the "Action" when the function is triggered.
  /// • >0: The "Action" is started by the trigger function with identical FollowID.
  /// • <0: The "Action" is stopped by the trigger function with identical FollowID.
  /// For more information see chapter 5.5.12.4 EmitterID, ListenerID, FollowID and OriginID
  OriginID           : DINT;  
  /// Relates to ListenerID >0
  /// Number of successful trigger -based command invocations
  /// For more information refer to chapter 5.5.12.4.
  InvocationCounter  : USINT;  
END_STRUCT
END_TYPE

// Library/POUs/SuperImposing/MC_MoveSuperImposed/Structures/MoveSuperImposedParCmd
{attribute 'pack_mode' := '1'} 
// ------------------------------------------------------------------------- 
//  SRCI Robot Library                                                
// ------------------------------------------------------------------------- 
//                                                                           
//  Object:      MoveSuperImposedParCmd                                       
//  Author:      Thorsten Brach                                                
//  Date:        2024-08-01
//
//  Description:                                              
//   
//                                                                           
//  Copyright: 
//    (C) 2024 Thorsten Brach. All rights reserved                                                                                                                                            
//             Licensed under the LGPL-3.0 license.
//                                                                           
//  Disclaimer:                                                                           
//    This project is provided without any guarantee and can be used for   
//    private and commercial purposes. Any use is at the user’s 
//    own risk and responsibility.
//
// -------------------------------------------------------------------------
TYPE MoveSuperImposedParCmd :
STRUCT
  /// Additional distance and orientation for superimposed positioning:
  Offset             : RobotCartesianPosition;
  /// Defines type of reference coordinate system of the offset position.
  ReferenceType      : ReferenceType;
  /// Value of the maximum velocity difference of the additional motion (not necessary reached).
  /// • > 0% Use specified value.
  /// • ≤ 0% Use the velocity defined by the move command that is superimposed. If no motion is active, use internal minimal velocity. (default)
 /// See chapter 5.5.7 Robot dynamics
  VelocityDiffRate   : REAL;
  /// Value of the maximum acceleration difference of the additional motion (not necessary reached).
  ///  •  <0% Use default acceleration (default)
  ///  •   0% Use internal minimal acceleration
  ///  • 100% Use maximal reference acceleration
  /// See chapter 5.5.7 Robot dynamics
  AccelerationDiffRate: REAL;
  /// Value of the maximum deceleration difference of the additional motion (not necessary reached).
  /// •  <0% Use default deceleration (default)
  /// •   0% Use internal minimal deceleration
  /// • 100% Use maximal reference deceleration
  /// See chapter 5.5.7 Robot dynamics
  DecelerationDiffRate: REAL;
  /// Value of the maximum jerk difference of the additional motion (not necessary reached).
  /// •  <0% Use default jerk (default) 
  /// •   0% Use internal minimal jerk
  /// • 100% Use maximal reference jerk
  /// See chapter 5.5.7 Robot dynamics
  JerkDiffRate        : REAL;
  /// Index of tool
  /// •      0: Flange (default)
  /// • 1..254: Tool frames
  ToolNo             : USINT;
  /// Index of frame
  /// •      0: WCS (default)
  /// • 1..254: User frames
  FrameNo            : USINT;
  /// ID of the trigger function that may be triggered:
  /// •  0: Immediately (default) - Start executing this function immediately.
  /// • >0: Trigger               - Start executing when the trigger function with the identical positive EmitterID is called
  ///                             - Stop executing when the trigger function with the identical negative EmitterID is called.
  /// For more information see chapter 5.5.12.4.
  ListenerID         : SINT;
  /// ID of Action that will be executed when this command is active
  /// • >0: Start Action - Start executing the Action function with the identical ListenerID.
  /// • <0: Stop Action  -  Stop executing the Action function with the identical ListenerID.
  /// • 0: No trigger (default)-  If no EmitterID is defined, the function will not trigger any Action during its execution
  /// For more information see section Triggers of this chapter or chapter 5.5.12.4.
  EmitterID          : ARRAY [0..3] OF SINT;  
END_STRUCT
END_TYPE

// Library/POUs/SuperImposing/MC_MoveSuperImposed/Structures/MoveSuperImposedRecvData
{attribute 'pack_mode' := '1'} 
// ------------------------------------------------------------------------- 
//  SRCI Robot Library                                                
// ------------------------------------------------------------------------- 
//                                                                           
//  Object:      MoveSuperImposedRecvData                                       
//  Author:      Thorsten Brach                                                
//  Date:        2024-08-01
//
//  Description:                                              
//   
//                                                                           
//  Copyright: 
//    (C) 2024 Thorsten Brach. All rights reserved                                                                                                                                            
//             Licensed under the LGPL-3.0 license.
//                                                                           
//  Disclaimer:                                                                           
//    This project is provided without any guarantee and can be used for   
//    private and commercial purposes. Any use is at the user’s 
//    own risk and responsibility.
//
// -------------------------------------------------------------------------
TYPE MoveSuperImposedRecvData EXTENDS RspHeader :
STRUCT
  /// Relates to ListenerID >0
  /// Number of successful trigger-based command invocations - For more information refer TO chapter 5.5.12.4
  InvocationCounter : USINT;  
  /// Reserve
  Reserve           : SINT;
  /// Unique system-generated ID of the "Action" when the function is triggered.
  /// • >0: The "Action" is started by the trigger funcrion with identical FollowID.
  /// • <0: The "Action" is stopped by the trigger function with identical FollowID.
  /// For more information see chapter 5.5.12.4 EmitterID, ListenerID, FollowID and OriginID
  OriginID          : INT;
  /// Percentage of already traversed distance of current job.
  /// If not supported : • -1
  Progress          : UINT;
  /// Distance-to-go of the current job.
  /// • -1: No valid value because move command is not yet active (valid values are pending) or not supported by RC
  /// • >0: Actual distance between current and target position
  /// •  0: Target position reached
  RemainingDistance  : REAL; 
END_STRUCT
END_TYPE

// Library/POUs/SuperImposing/MC_MoveSuperImposed/Structures/MoveSuperImposedSendData
{attribute 'pack_mode' := '1'}
// ------------------------------------------------------------------------- 
//  SRCI Robot Library                                                
// ------------------------------------------------------------------------- 
//                                                                           
//  Object:      MoveSuperImposedSendData                                       
//  Author:      Thorsten Brach                                                
//  Date:        2024-08-01
//
//  Description:                                              
//   
//                                                                           
//  Copyright: 
//    (C) 2024 Thorsten Brach. All rights reserved                                                                                                                                            
//             Licensed under the LGPL-3.0 license.
//                                                                           
//  Disclaimer:                                                                           
//    This project is provided without any guarantee and can be used for   
//    private and commercial purposes. Any use is at the user’s 
//    own risk and responsibility.
//
// -------------------------------------------------------------------------
TYPE MoveSuperImposedSendData EXTENDS CmdHeader: 
STRUCT
  /// ID of Action that will be executed when this command is active
  /// • >0: Start Action - Start executing the Action function with the identical ListenerID.
  /// • <0: Stop Action  -  Stop executing the Action function with the identical ListenerID.
  /// • 0: No trigger (default)-  If no EmitterID is defined, the function will not trigger any Action during its execution
  /// For more information see section Triggers of this chapter or chapter 5.5.12.4.
  EmitterID          : ARRAY [0..3] OF SINT;
  /// ID of the trigger function that may be triggered:
  /// • 0: Immediately (default). - Start executing THIS function immediately.
  /// • >0: Triggero Start executing when the trigger function with the identical EmitterID is called.
  /// For more information see chapter 5.5.12.4.
  ListenerID         : SINT;
  /// Reserve
  Reserve            : BYTE;
  /// Value of the maximum velocity difference of the additional motion (not necessary reached).
  /// • > 0% Use specified value.
  /// • ≤ 0% Use the velocity defined by the move command that is superimposed. If no motion is active, use internal minimal velocity. (default)
 /// See chapter 5.5.7 Robot dynamics
  VelocityDiffRate   : UINT;
  /// Value of the maximum acceleration difference of the additional motion (not necessary reached).
  ///  •  <0% Use default acceleration (default)
  ///  •   0% Use internal minimal acceleration
  ///  • 100% Use maximal reference acceleration
  /// See chapter 5.5.7 Robot dynamics
  AccelerationDiffRate: UINT;
  /// Value of the maximum deceleration difference of the additional motion (not necessary reached).
  /// •  <0% Use default deceleration (default)
  /// •   0% Use internal minimal deceleration
  /// • 100% Use maximal reference deceleration
  /// See chapter 5.5.7 Robot dynamics
  DecelerationDiffRate: UINT;
  /// Value of the maximum jerk difference of the additional motion (not necessary reached).
  /// •  <0% Use default jerk (default) 
  /// •   0% Use internal minimal jerk
  /// • 100% Use maximal reference jerk
  /// See chapter 5.5.7 Robot dynamics
  JerkDiffRate        : UINT;
  /// Index of tool
  /// •      0: Flange (default)
  /// • 1..254: Tool frames
  ToolNo             : USINT;
  /// Index of frame
  /// •      0: WCS (default)
  /// • 1..254: User frames
  FrameNo            : USINT;
  /// Additional distance and orientation for superimposed positioning:
  Offset             : RobotCartesianPosition;
  /// Defines type of reference coordinate system of the offset position
  ReferenceType      : USINT;
  /// Reserve2
  Reserve2           : BYTE;  
END_STRUCT
END_TYPE

// Library/POUs/SuperImposing/MC_MoveSuperImposedDynamic/Structures/MoveSuperImposedDynamicOutCmd
{attribute 'pack_mode' := '1'} 
// ------------------------------------------------------------------------- 
//  SRCI Robot Library                                                
// ------------------------------------------------------------------------- 
//                                                                           
//  Object:      MoveSuperImposedDynamicOutCmd                                       
//  Author:      Thorsten Brach                                                
//  Date:        2024-08-01
//
//  Description:                                              
//   
//                                                                           
//  Copyright: 
//    (C) 2024 Thorsten Brach. All rights reserved                                                                                                                                            
//             Licensed under the LGPL-3.0 license.
//                                                                           
//  Disclaimer:                                                                           
//    This project is provided without any guarantee and can be used for   
//    private and commercial purposes. Any use is at the user’s 
//    own risk and responsibility.
//
// -------------------------------------------------------------------------
TYPE MoveSuperImposedDynamicOutCmd :
STRUCT
  /// Distance-to-go [mm] of the current job
  /// • -1: No valid value because move command is not yet active (valid values are pending) or not supported by RC
  /// • >0: Actual distance between current and target position
  /// •  0: Target position reached
  RemainingDistance  : REAL;
  /// Percentage of already traversed superimposed offset.
  /// If not supported : • -1
  Progress           : REAL;
  /// TRUE if the offset for superimposed positioning is reached.
  OffsetReached      : BOOL;
END_STRUCT
END_TYPE

// Library/POUs/SuperImposing/MC_MoveSuperImposedDynamic/Structures/MoveSuperImposedDynamicParCmd
{attribute 'pack_mode' := '1'} 
// ------------------------------------------------------------------------- 
//  SRCI Robot Library                                                
// ------------------------------------------------------------------------- 
//                                                                           
//  Object:      MoveSuperImposedDynamicParCmd                                       
//  Author:      Thorsten Brach                                                
//  Date:        2024-08-01
//
//  Description:                                              
//   
//                                                                           
//  Copyright: 
//    (C) 2024 Thorsten Brach. All rights reserved                                                                                                                                            
//             Licensed under the LGPL-3.0 license.
//                                                                           
//  Disclaimer:                                                                           
//    This project is provided without any guarantee and can be used for   
//    private and commercial purposes. Any use is at the user’s 
//    own risk and responsibility.
//
// -------------------------------------------------------------------------
TYPE MoveSuperImposedDynamicParCmd :
STRUCT
  /// Additional distance and orientation for superimposed positioning
  Offset             : RobotCartesianPosition;
  /// Defines type of reference coordinate system of the offset position.
  ReferenceType      : ReferenceType;
  /// Value of the maximum velocity difference of the additional motion (not necessary reached).
  /// • > 0% Use specified value.
  /// • ≤ 0% Use the velocity defined by the move command that is superimposed. If no motion is active, use internal minimal velocity. (default)
 /// See chapter 5.5.7 Robot dynamics
  VelocityDiffRate   : REAL;
  /// Value of the maximum acceleration difference of the additional motion (not necessary reached).
  ///  •  <0% Use default acceleration (default)
  ///  •   0% Use internal minimal acceleration
  ///  • 100% Use maximal reference acceleration
  /// See chapter 5.5.7 Robot dynamics
  AccelerationDiffRate: REAL;
  /// Value of the maximum deceleration difference of the additional motion (not necessary reached).
  /// •  <0% Use default deceleration (default)
  /// •   0% Use internal minimal deceleration
  /// • 100% Use maximal reference deceleration
  /// See chapter 5.5.7 Robot dynamics
  DecelerationDiffRate: REAL;
  /// Value of the maximum jerk difference of the additional motion (not necessary reached).
  /// •  <0% Use default jerk (default) 
  /// •   0% Use internal minimal jerk
  /// • 100% Use maximal reference jerk
  /// See chapter 5.5.7 Robot dynamics
  JerkDiffRate        : REAL;
  /// Index of tool
  /// •      0: Flange (default)
  /// • 1..254: Tool frames
  ToolNo             : USINT;
  /// Index of frame
  /// •      0: WCS (default)
  /// • 1..254: User frames
  FrameNo            : USINT;
  /// Define the interpolation mode for the superimposed motion
  InterpolationMode  : InterpolationMode;
END_STRUCT
END_TYPE

// Library/POUs/SuperImposing/MC_MoveSuperImposedDynamic/Structures/MoveSuperImposedDynamicRecvData
{attribute 'pack_mode' := '1'} 
// ------------------------------------------------------------------------- 
//  SRCI Robot Library                                                
// ------------------------------------------------------------------------- 
//                                                                           
//  Object:      MoveSuperImposedDynamicRecvData                                       
//  Author:      Thorsten Brach                                                
//  Date:        2024-08-01
//
//  Description:                                              
//   
//                                                                           
//  Copyright: 
//    (C) 2024 Thorsten Brach. All rights reserved                                                                                                                                            
//             Licensed under the LGPL-3.0 license.
//                                                                           
//  Disclaimer:                                                                           
//    This project is provided without any guarantee and can be used for   
//    private and commercial purposes. Any use is at the user’s 
//    own risk and responsibility.
//
// -------------------------------------------------------------------------
TYPE MoveSuperImposedDynamicRecvData EXTENDS RspHeader :
STRUCT
  /// Percentage of already traversed distance of current job.
  /// If not supported : • -1
  Progress          : UINT;
  /// Distance-to-go of the current job.
  /// • -1: No valid value because move command is not yet active (valid values are pending) or not supported by RC
  /// • >0: Actual distance between current and target position
  /// •  0: Target position reached
  RemainingDistance  : REAL;
  /// TRUE if the offset for superimposed positioning is reached.
  OffsetReached      : BOOL;  
END_STRUCT
END_TYPE

// Library/POUs/SuperImposing/MC_MoveSuperImposedDynamic/Structures/MoveSuperImposedDynamicSendData
{attribute 'pack_mode' := '1'}
// ------------------------------------------------------------------------- 
//  SRCI Robot Library                                                
// ------------------------------------------------------------------------- 
//                                                                           
//  Object:      MoveSuperImposedDynamicSendData                                       
//  Author:      Thorsten Brach                                                
//  Date:        2024-08-01
//
//  Description:                                              
//   
//                                                                           
//  Copyright: 
//    (C) 2024 Thorsten Brach. All rights reserved                                                                                                                                            
//             Licensed under the LGPL-3.0 license.
//                                                                           
//  Disclaimer:                                                                           
//    This project is provided without any guarantee and can be used for   
//    private and commercial purposes. Any use is at the user’s 
//    own risk and responsibility.
//
// -------------------------------------------------------------------------
TYPE MoveSuperImposedDynamicSendData EXTENDS CmdHeader: 
STRUCT
  /// Value of the maximum velocity difference of the additional motion (not necessary reached).
  /// • > 0% Use specified value.
  /// • ≤ 0% Use the velocity defined by the move command that is superimposed. If no motion is active, use internal minimal velocity. (default)
 /// See chapter 5.5.7 Robot dynamics
  VelocityDiffRate    : UINT;
  /// Value of the maximum acceleration difference of the additional motion (not necessary reached).
  ///  •  <0% Use default acceleration (default)
  ///  •   0% Use internal minimal acceleration
  ///  • 100% Use maximal reference acceleration
  /// See chapter 5.5.7 Robot dynamics
  AccelerationDiffRate: UINT;
  /// Value of the maximum deceleration difference of the additional motion (not necessary reached).
  /// •  <0% Use default deceleration (default)
  /// •   0% Use internal minimal deceleration
  /// • 100% Use maximal reference deceleration
  /// See chapter 5.5.7 Robot dynamics
  DecelerationDiffRate: UINT;
  /// Value of the maximum jerk difference of the additional motion (not necessary reached).
  /// •  <0% Use default jerk (default) 
  /// •   0% Use internal minimal jerk
  /// • 100% Use maximal reference jerk
  /// See chapter 5.5.7 Robot dynamics
  JerkDiffRate        : UINT;
  /// Index of tool
  /// •      0: Flange (default)
  /// • 1..254: Tool frames
  ToolNo              : USINT;
  /// Index of frame
  /// •      0: WCS (default)
  /// • 1..254: User frames
  FrameNo             : USINT;
  /// Reserve X
  Reserve_X           : REAL;
  /// Additional distance and orientation for superimposed positioning
  Offset              : RobotCartesianPosition;
  /// Defines type of reference coordinate system of the offset position.
  ReferenceType       : USINT;
  /// Define the interpolation mode for the superimposed motion
  InterpolationMode   : USINT;
END_STRUCT
END_TYPE

// Library/POUs/Trigger/MC_ReactAtTrigger/Structures/ReactAtTriggerOutCmd
{attribute 'pack_mode' := '1'} 
// ------------------------------------------------------------------------- 
//  SRCI Robot Library                                                
// ------------------------------------------------------------------------- 
//                                                                           
//  Object:      ReactAtTriggerOutCmd                                       
//  Author:      Thorsten Brach                                                
//  Date:        2024-08-03
//
//  Description:                                              
//   
//                                                                           
//  Copyright: 
//    (C) 2024 Thorsten Brach. All rights reserved                                                                                                                                            
//             Licensed under the LGPL-3.0 license.
//                                                                           
//  Disclaimer:                                                                           
//    This project is provided without any guarantee and can be used for   
//    private and commercial purposes. Any use is at the user’s 
//    own risk and responsibility.
//
// -------------------------------------------------------------------------
TYPE ReactAtTriggerOutCmd :
STRUCT
  /// Unique system-generated ID of the "Action" when the function is triggered.
  /// • >0: The "Action" is started by the trigger function with identical FollowID.
  /// • <0: The "Action" is stopped by the trigger function with identical FollowID.
  /// For more information see chapter 5.5.12.4 EmitterID, ListenerID, FollowID and OriginID
  OriginID               : INT;
  /// Relates to ListenerID >0
  /// Number of successful trigger -based command invocations
  /// For more information refer to chapter 5.5.12.4.
  InvocationCounter      : USINT;
END_STRUCT
END_TYPE

// Library/POUs/Trigger/MC_ReactAtTrigger/Structures/ReactAtTriggerParCmd
{attribute 'pack_mode' := '1'} 
// ------------------------------------------------------------------------- 
//  SRCI Robot Library                                                
// ------------------------------------------------------------------------- 
//                                                                           
//  Object:      ReactAtTriggerParCmd                                       
//  Author:      Thorsten Brach                                                
//  Date:        2024-08-03
//
//  Description:                                              
//   
//                                                                           
//  Copyright: 
//    (C) 2024 Thorsten Brach. All rights reserved                                                                                                                                            
//             Licensed under the LGPL-3.0 license.
//                                                                           
//  Disclaimer:                                                                           
//    This project is provided without any guarantee and can be used for   
//    private and commercial purposes. Any use is at the user’s 
//    own risk and responsibility.
//
// -------------------------------------------------------------------------
TYPE ReactAtTriggerParCmd :
STRUCT
  /// Defines RC’s and robot’s behavior when the"Action" is executed.
  ReactionMode           : TriggerReactionMode;
  /// ID of associated trigger function:
  /// • 0: Immediately (default) - Start executing this function immediately.
  /// • >0: Trigger -  Start executing, when the trigger function with the identical EmitterID is triggered.
  /// Always positive.
  /// For more information, see chapter 5.5.12 Triggers
  ListenerID             : SINT;
END_STRUCT
END_TYPE

// Library/POUs/Trigger/MC_ReactAtTrigger/Structures/ReactAtTriggerRecvData
{attribute 'pack_mode' := '1'} 
// ------------------------------------------------------------------------- 
//  SRCI Robot Library                                                
// ------------------------------------------------------------------------- 
//                                                                           
//  Object:      ReactAtTriggerRecvData                                       
//  Author:      Thorsten Brach                                                
//  Date:        2024-08-03
//
//  Description:                                              
//   
//                                                                           
//  Copyright: 
//    (C) 2024 Thorsten Brach. All rights reserved                                                                                                                                            
//             Licensed under the LGPL-3.0 license.
//                                                                           
//  Disclaimer:                                                                           
//    This project is provided without any guarantee and can be used for   
//    private and commercial purposes. Any use is at the user’s 
//    own risk and responsibility.
//
// -------------------------------------------------------------------------
TYPE ReactAtTriggerRecvData EXTENDS RspHeader :
STRUCT
  /// Relates to ListenerID >0
  /// Number of successful trigger-based command invocations - For more information refer TO chapter 5.5.12.4
  InvocationCounter : USINT;  
  /// Reserve
  Reserve           : SINT;
  /// Unique system-generated ID of the "Action" when the function is triggered.
  /// • >0: The "Action" is started by the trigger funcrion with identical FollowID.
  /// • <0: The "Action" is stopped by the trigger function with identical FollowID.
  /// For more information see chapter 5.5.12.4 EmitterID, ListenerID, FollowID and OriginID
  OriginID          : INT;
END_STRUCT
END_TYPE

// Library/POUs/Trigger/MC_ReactAtTrigger/Structures/ReactAtTriggerSendData
{attribute 'pack_mode' := '1'}
// ------------------------------------------------------------------------- 
//  SRCI Robot Library                                                
// ------------------------------------------------------------------------- 
//                                                                           
//  Object:      ReactAtTriggerSendData                                       
//  Author:      Thorsten Brach                                                
//  Date:        2024-08-03
//
//  Description:                                              
//   
//                                                                           
//  Copyright: 
//    (C) 2024 Thorsten Brach. All rights reserved                                                                                                                                            
//             Licensed under the LGPL-3.0 license.
//                                                                           
//  Disclaimer:                                                                           
//    This project is provided without any guarantee and can be used for   
//    private and commercial purposes. Any use is at the user’s 
//    own risk and responsibility.
//
// -------------------------------------------------------------------------
TYPE ReactAtTriggerSendData EXTENDS CmdHeader: 
STRUCT
  /// ID of Action that will be executed when this command is active
  /// • >0: Start Action - Start executing the Action function with the identical ListenerID.
  /// • <0: Stop Action  -  Stop executing the Action function with the identical ListenerID.
  /// • 0: No trigger (default)-  If no EmitterID is defined, the function will not trigger any Action during its execution
  /// For more information see section Triggers of this chapter or chapter 5.5.12.4.
  EmitterID          : ARRAY [0..3] OF SINT;  
  /// ID of associated trigger function:
  /// • 0: Immediately (default) - Start executing this function immediately.
  /// • >0: Trigger -  Start executing, when the trigger function with the identical EmitterID is triggered.
  /// Always positive.
  /// For more information, see chapter 5.5.12 Triggers
  ListenerID         : SINT;
  /// Reserve
  Reserve            : SINT;
  /// Defines RC’s and robot’s behavior when the"Action" is executed.
  ReactionMode       : TriggerReactionMode;
END_STRUCT
END_TYPE

// Library/POUs/Trigger/MC_SetTriggerError/Structures/SetTriggerErrorOutCmd
{attribute 'pack_mode' := '1'} 
// ------------------------------------------------------------------------- 
//  SRCI Robot Library                                                
// ------------------------------------------------------------------------- 
//                                                                           
//  Object:      SetTriggerErrorOutCmd                                       
//  Author:      Thorsten Brach                                                
//  Date:        2024-08-03
//
//  Description:                                              
//   
//                                                                           
//  Copyright: 
//    (C) 2024 Thorsten Brach. All rights reserved                                                                                                                                            
//             Licensed under the LGPL-3.0 license.
//                                                                           
//  Disclaimer:                                                                           
//    This project is provided without any guarantee and can be used for   
//    private and commercial purposes. Any use is at the user’s 
//    own risk and responsibility.
//
// -------------------------------------------------------------------------
TYPE SetTriggerErrorOutCmd :
STRUCT
  /// Unique system-generated ID of the "Action" when the function is triggered.
  /// • >0: The "Action" is started by the trigger function with identical FollowID.
  /// • <0: The "Action" is stopped by the trigger function with identical FollowID.
  /// For more information see chapter 5.5.12.4 EmitterID, ListenerID, FollowID and OriginID
  OriginID               : INT;
  /// Relates to ListenerID >0
  /// Number of successful trigger -based command invocations
  /// For more information refer to chapter 5.5.12.4.
  InvocationCounter      : USINT;
  /// Unique system-generated ID of the trigger function when the function is called by user.
  /// For more information see chapter 5.5.12.4.
  FollowID               : DINT;  
END_STRUCT
END_TYPE

// Library/POUs/Trigger/MC_SetTriggerError/Structures/SetTriggerErrorParCmd
{attribute 'pack_mode' := '1'} 
// ------------------------------------------------------------------------- 
//  SRCI Robot Library                                                
// ------------------------------------------------------------------------- 
//                                                                           
//  Object:      SetTriggerErrorParCmd                                       
//  Author:      Thorsten Brach                                                
//  Date:        2024-08-03
//
//  Description:                                              
//   
//                                                                           
//  Copyright: 
//    (C) 2024 Thorsten Brach. All rights reserved                                                                                                                                            
//             Licensed under the LGPL-3.0 license.
//                                                                           
//  Disclaimer:                                                                           
//    This project is provided without any guarantee and can be used for   
//    private and commercial purposes. Any use is at the user’s 
//    own risk and responsibility.
//
// -------------------------------------------------------------------------
TYPE SetTriggerErrorParCmd :
STRUCT
  /// Defines error origin through which the associated Action will be triggered
  Mode                   : ErrorTriggerMode;
  /// Defines message codes through which the associated Action will be triggered (relates to Mode 6 and 7)
  MessageCodes           : ARRAY [0..RobotLibraryParameter.MESSAGE_CODES_MAX] OF DWORD;
  /// Defines if parametrization messages are included (relates to Mode 0 to 5)
  /// • FALSE (default): Do not include incorrect parametrization
  /// • TRUE: Include incorrect parametrization
  IncludeParameterValidation : BOOL;
  /// ID of associated trigger function:
  /// • 0: Immediately (default) - Start executing this function immediately.
  /// • >0: Trigger -  Start executing, when the trigger function with the identical EmitterID is triggered.
  /// Always positive.
  /// For more information, see chapter 5.5.12 Triggers
  ListenerID             : SINT;
  /// ID of the Action function that will be executed when the trigger condition is met
  /// • >0: Start Action        - Start executing the Action function with the identical ListenerID.
  /// • <0: Stop Action         - Stop executing the Action function with the identical ListenerID.
  /// •  0: Undefined (default) - If no EmitterID is defined, the function returns an error message
  /// For more information see chapter 5.5.12.4
  EmitterID              : SINT;  
END_STRUCT
END_TYPE

